// TIA Portal V18 export
TYPE "MEStoPLC_SubCheckIn_ext"
// stored: IsFailsafeCompliant false
   STRUCT
      Spare : Byte;   // SpareByte
      Load_SubPart1OK : Bool;   // 子零件可用标志位,收到MES.SubPartReqMesDone后开始使用
      Load_SubPart1tNG : Bool;   // 子零件禁用标志位,收到MES.SubPartReqMesDone后弃料
      Load_SubPart1ReqMesDone : Bool;   // 查询完成,PLC复位PLC.Load_SubPart*ChickInReq
      SubPart1Spare : Bool;   // Spare
      SubPart1Spare1 : Bool;   // Spare
      SubPart1Spare2 : Bool;   // Spare
      SubPart1Spare3 : Bool;   // Spare
      SubPart1Spare4 : Bool;   // Spare
      Load_SubPart2OK : Bool;   // 子零件可用标志位,收到MES.SubPartReqMesDone后开始使用
      Load_SubPart2tNG : Bool;   // 子零件禁用标志位,收到MES.SubPartReqMesDone后弃料
      Load_SubPart2ReqMesDone : Bool;   // 查询完成,PLC复位PLC.Load_SubPart*ChickInReq
      SubPart2Spare : Bool;   // Spare
      SubPart2Spare1 : Bool;   // Spare
      SubPart2Spare2 : Bool;   // Spare
      SubPart2Spare3 : Bool;   // Spare
      SubPart2Spare4 : Bool;   // Spare
      Load_SubPart3OK : Bool;   // 子零件可用标志位,收到MES.SubPartReqMesDone后开始使用
      Load_SubPart3tNG : Bool;   // 子零件禁用标志位,收到MES.SubPartReqMesDone后弃料
      Load_SubPart3ReqMesDone : Bool;   // 查询完成,PLC复位PLC.Load_SubPart*ChickInReq
      SubPart3Spare : Bool;   // Spare
      SubPart3Spare1 : Bool;   // Spare
      SubPart3Spare2 : Bool;   // Spare
      SubPart3Spare3 : Bool;   // Spare
      SubPart3Spare4 : Bool;   // Spare
      Load_SubPart4OK : Bool;   // 子零件可用标志位,收到MES.SubPartReqMesDone后开始使用
      Load_SubPart4tNG : Bool;   // 子零件禁用标志位,收到MES.SubPartReqMesDone后弃料
      Load_SubPart4ReqMesDone : Bool;   // 查询完成,PLC复位PLC.Load_SubPart*ChickInReq
      SubPart4Spare : Bool;   // Spare
      SubPart4Spare1 : Bool;   // Spare
      SubPart4Spare2 : Bool;   // Spare
      SubPart4Spare3 : Bool;   // Spare
      SubPart4Spare4 : Bool;   // Spare
      Load_SubPart5OK : Bool;   // 子零件可用标志位,收到MES.SubPartReqMesDone后开始使用
      Load_SubPart5tNG : Bool;   // 子零件禁用标志位,收到MES.SubPartReqMesDone后弃料
      Load_SubPart5ReqMesDone : Bool;   // 查询完成,PLC复位PLC.Load_SubPart*ChickInReq
      SubPart5Spare : Bool;   // Spare
      SubPart5Spare1 : Bool;   // Spare
      SubPart5Spare2 : Bool;   // Spare
      SubPart5Spare3 : Bool;   // Spare
      SubPart5Spare4 : Bool;   // Spare
      Load_SubPart6OK : Bool;   // 子零件可用标志位,收到MES.SubPartReqMesDone后开始使用
      Load_SubPart6tNG : Bool;   // 子零件禁用标志位,收到MES.SubPartReqMesDone后弃料
      Load_SubPart6ReqMesDone : Bool;   // 查询完成,PLC复位PLC.Load_SubPart*ChickInReq
      SubPart6Spare : Bool;   // Spare
      SubPart6Spare1 : Bool;   // Spare
      SubPart6Spare2 : Bool;   // Spare
      SubPart6Spare3 : Bool;   // Spare
      SubPart6Spare4 : Bool;   // Spare
      Load_SubPart7OK : Bool;   // 子零件可用标志位,收到MES.SubPartReqMesDone后开始使用
      Load_SubPart7tNG : Bool;   // 子零件禁用标志位,收到MES.SubPartReqMesDone后弃料
      Load_SubPart7ReqMesDone : Bool;   // 查询完成,PLC复位PLC.Load_SubPart*ChickInReq
      SubPart7Spare : Bool;   // Spare
      SubPart7Spare1 : Bool;   // Spare
      SubPart7Spare2 : Bool;   // Spare
      SubPart7Spare3 : Bool;   // Spare
      SubPart7Spare4 : Bool;   // Spare
      Load_SubPart8OK : Bool;   // 子零件可用标志位,收到MES.SubPartReqMesDone后开始使用
      Load_SubPart8tNG : Bool;   // 子零件禁用标志位,收到MES.SubPartReqMesDone后弃料
      Load_SubPart8ReqMesDone : Bool;   // 查询完成,PLC复位PLC.Load_SubPart*ChickInReq
      SubPart8Spare : Bool;   // Spare
      SubPart8Spare1 : Bool;   // Spare
      SubPart8Spare2 : Bool;   // Spare
      SubPart8Spare3 : Bool;   // Spare
      SubPart8Spare4 : Bool;   // Spare
      SpareByte : Byte;   // SpareByte
   END_STRUCT;
END_TYPE
